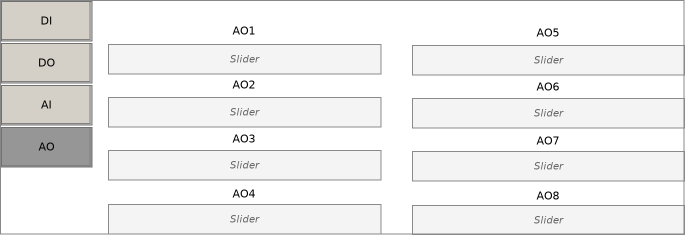
VISUALIZATION Analog_Outputs  // 685x235
    Slider (108,44 273x30), variable: GVL_IO.AO1, scale 4..20
    Slider (108,97 273x30), variable: GVL_IO.AO2, scale 4..20
    Slider (108,150 273x30), variable: GVL_IO.AO3, scale 4..20
    Slider (108,204 273x30), variable: GVL_IO.AO4, scale 4..20
    Slider (412,45 273x30), variable: GVL_IO.AO5, scale 4..20
    Slider (412,98 273x30), variable: GVL_IO.AO6, scale 4..20
    Slider (412,151 273x30), variable: GVL_IO.AO7, scale 4..20
    Slider (412,205 273x30), variable: GVL_IO.AO8, scale 4..20
    Label (169,16 150x30), "AO1"
    Label (169,70 150x30), "AO2"
    Label (169,124 150x30), "AO3"
    Label (169,179 150x30), "AO4"
    Label (473,18 150x30), "AO5"
    Label (473,72 150x30), "AO6"
    Label (473,126 150x30), "AO7"
    Label (473,181 150x30), "AO8"
    Button (1,127 91x40), "AO"
        OnMouseUp: change screen: Analog_Outputs
    Button (1,1 91x40), "DI"
        OnMouseUp: change screen: Digital_Inputs
    Button (1,43 91x40), "DO"
        OnMouseDown: change screen: Digital_Outputs
        OnMouseUp: change screen: Digital_Outputs
    Button (1,85 91x40), "AI"
        OnMouseUp: change screen: Analog_Inputs
END_VISUALIZATION

(* stored: Version 1.1.0.1, ProductVersion 3.1.4024.4
   Visu Analog_Outputs: Id {fa74690f-1bc4-4df7-b15c-a982dc1d41a9} *)
